(* CODESYS project opas-OCFB_IN-test-project

Project tree, tasks and I/O mapping:
  Device : CODESYS Control Win V3 x64, 3S - Smart Software Solutions GmbH, version 3.5.19.10
    application Application
      libraries: Standard, 3.5.18.0 (System); OPAS OCF Library, 1.0.0.0 (CODESYS Corporation)
      task MainTask (cyclic, interval t#20ms, priority 1) calls PLC_PRG
      program OCFBs [LD]
      program OCFBs_sim [LD]
      program PLC_PRG [ST]
      Sandbox/
        function block FB_FINAL_TEST [ST]
      SIM/
      visualisation Visualization
    SoftMotion General Axis Pool : SoftMotion General Axis Pool, 3S - Smart Software Solutions GmbH, version 4.11.0.0
    SoftMotion General Axis Pool : SoftMotion General Axis Pool, 3S - Smart Software Solutions GmbH, version 4.11.0.0
  text list GlobalTextList
*)

// Device/Application/PLC_PRG
PROGRAM PLC_PRG
VAR
	xAddConnection : BOOL;
	myAliasServerConnection : org_opengroup_opas_OCF.AliasServerConnection;
	fbFinal1 : FB_FINAL_TEST;
	fbFinal2 : FB_FINAL_TEST;
END_VAR

//OCFBs_sim();
OCFBs();

END_PROGRAM

// Device/Application/OCFBs_sim
PROGRAM OCFBs_sim
VAR
	xEnableAll : bool := true;
	tag1_OCFB_IN_SIM: org_opengroup_opas_OCF.OCFB_IN_SIM;
	tag2_OCFB_IN_SIM: org_opengroup_opas_OCF.OCFB_IN_SIM;
	tag3_OCFB_IN_SIM: org_opengroup_opas_OCF.OCFB_IN_SIM;
	tag4_OCFB_IN_SIM: org_opengroup_opas_OCF.OCFB_IN_SIM;
	tag5_OCFB_IN_SIM: org_opengroup_opas_OCF.OCFB_IN_SIM;
	tag6_OCFB_IN_SIM: org_opengroup_opas_OCF.OCFB_IN_SIM;
	tag7_OCFB_IN_SIM: org_opengroup_opas_OCF.OCFB_IN_SIM;
	
	xUtil1 : BOOL;
	xUtil2 : BOOL;
	xUtil3 : BOOL;
	xUtil4 : BOOL;
	iCount: UDINT;
END_VAR

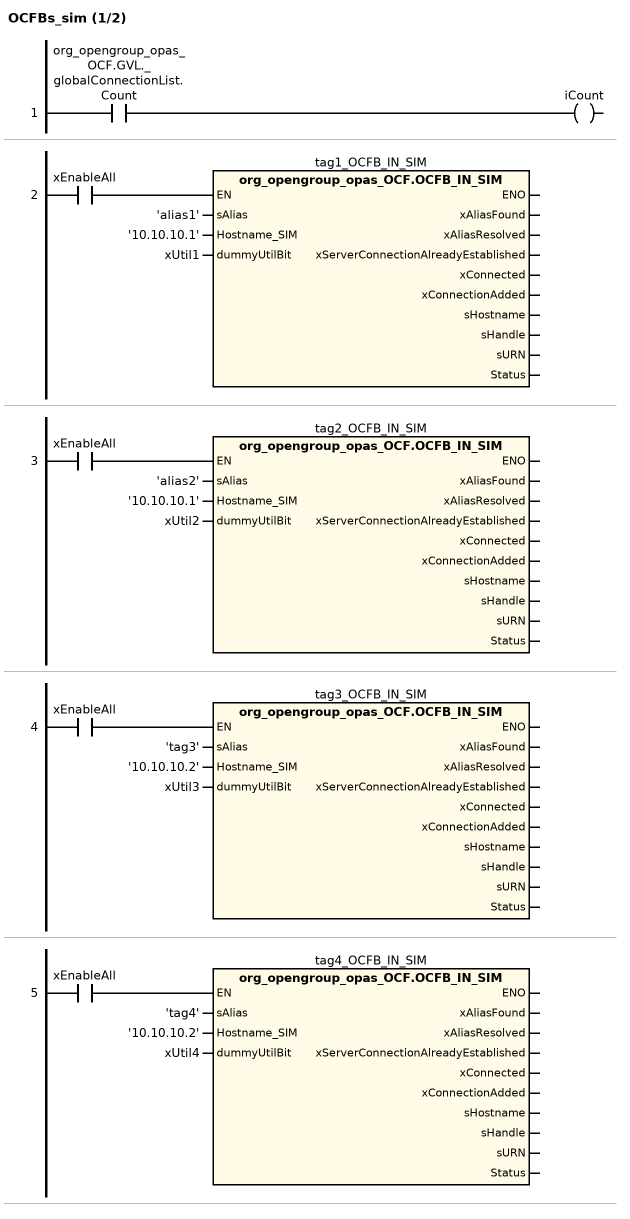
// NETWORK 1
iCount := org_opengroup_opas_OCF.GVL._globalConnectionList.Count;

// NETWORK 2
IF xEnableAll THEN
    tag1_OCFB_IN_SIM(sAlias := 'alias1', Hostname_SIM := '10.10.10.1', dummyUtilBit := xUtil1); // org_opengroup_opas_OCF.OCFB_IN_SIM
END_IF

// NETWORK 3
IF xEnableAll THEN
    tag2_OCFB_IN_SIM(sAlias := 'alias2', Hostname_SIM := '10.10.10.1', dummyUtilBit := xUtil2); // org_opengroup_opas_OCF.OCFB_IN_SIM
END_IF

// NETWORK 4
IF xEnableAll THEN
    tag3_OCFB_IN_SIM(sAlias := 'tag3', Hostname_SIM := '10.10.10.2', dummyUtilBit := xUtil3); // org_opengroup_opas_OCF.OCFB_IN_SIM
END_IF

// NETWORK 5
IF xEnableAll THEN
    tag4_OCFB_IN_SIM(sAlias := 'tag4', Hostname_SIM := '10.10.10.2', dummyUtilBit := xUtil4); // org_opengroup_opas_OCF.OCFB_IN_SIM
END_IF

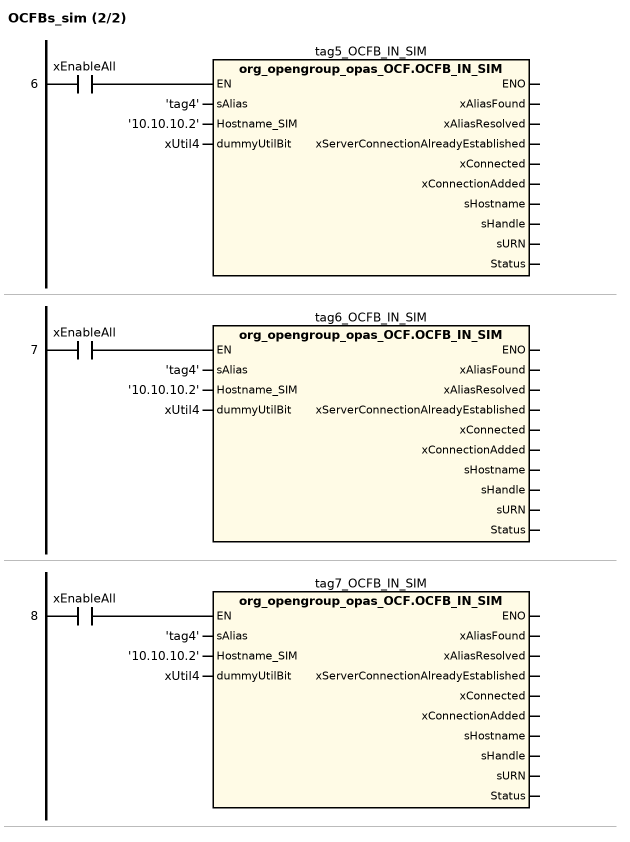
// NETWORK 6
IF xEnableAll THEN
    tag5_OCFB_IN_SIM(sAlias := 'tag4', Hostname_SIM := '10.10.10.2', dummyUtilBit := xUtil4); // org_opengroup_opas_OCF.OCFB_IN_SIM
END_IF

// NETWORK 7
IF xEnableAll THEN
    tag6_OCFB_IN_SIM(sAlias := 'tag4', Hostname_SIM := '10.10.10.2', dummyUtilBit := xUtil4); // org_opengroup_opas_OCF.OCFB_IN_SIM
END_IF

// NETWORK 8
IF xEnableAll THEN
    tag7_OCFB_IN_SIM(sAlias := 'tag4', Hostname_SIM := '10.10.10.2', dummyUtilBit := xUtil4); // org_opengroup_opas_OCF.OCFB_IN_SIM
END_IF

END_PROGRAM

// Device/Application/OCFBs
PROGRAM OCFBs
VAR
	xEnableAll : bool := true;
	tag1_OCFB_IN_SIM: org_opengroup_opas_OCF.OCFB_IN_LREAL;
	tag2_OCFB_IN_SIM: org_opengroup_opas_OCF.OCFB_IN_LREAL;
	//tag3_OCFB_IN_SIM: org_opengroup_opas_OCF.OCFB_IN_LREAL;
	//tag4_OCFB_IN_SIM: org_opengroup_opas_OCF.OCFB_IN_LREAL;
	//tag5_OCFB_IN_SIM: org_opengroup_opas_OCF.OCFB_IN_LREAL;
	//tag6_OCFB_IN_SIM: org_opengroup_opas_OCF.OCFB_IN_LREAL;
	//tag7_OCFB_IN_SIM: org_opengroup_opas_OCF.OCFB_IN_LREAL;
	
	xUtil1 : BOOL;
	xUtil2 : BOOL;
	xUtil3 : BOOL;
	xUtil4 : BOOL;
	iCount: UDINT;
	bEnable1: BOOL;
	bEnable2: BOOL;
END_VAR

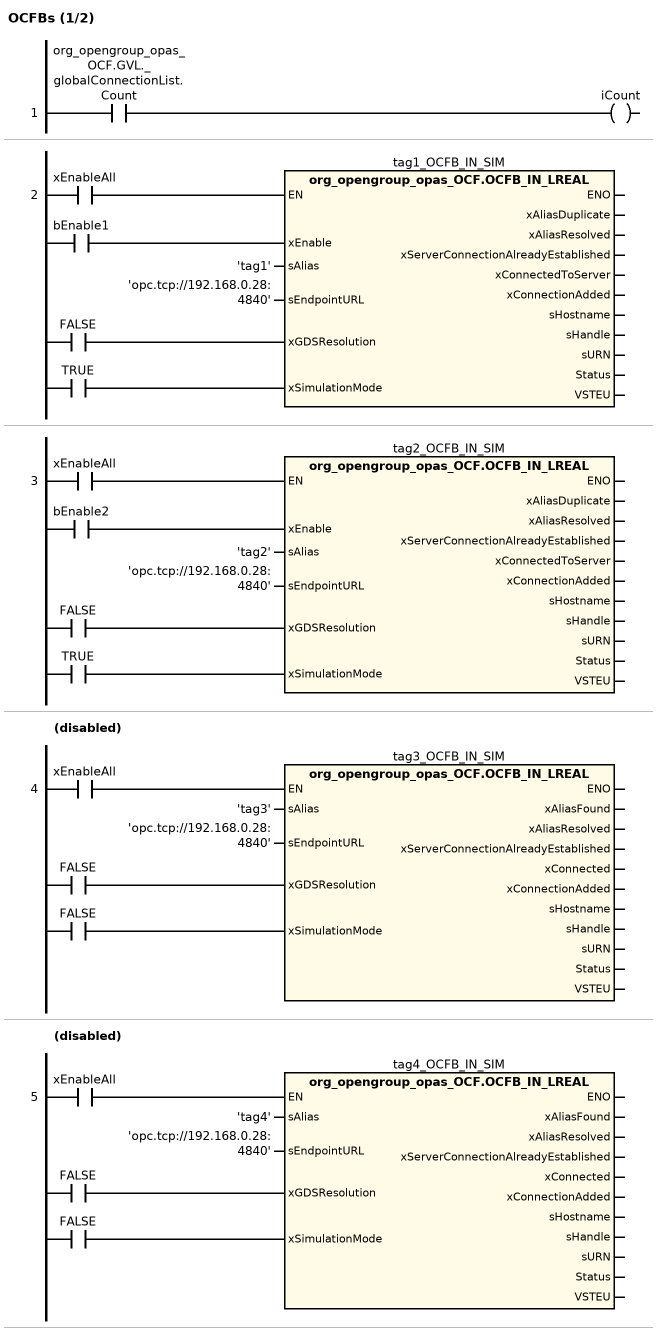
// NETWORK 1
iCount := org_opengroup_opas_OCF.GVL._globalConnectionList.Count;

// NETWORK 2
IF xEnableAll THEN
    tag1_OCFB_IN_SIM(
        xEnable := bEnable1,
        sAlias := 'tag1',
        sEndpointURL := 'opc.tcp://192.168.0.28:4840',
        xGDSResolution := FALSE,
        xSimulationMode := TRUE); // org_opengroup_opas_OCF.OCFB_IN_LREAL
END_IF

// NETWORK 3
IF xEnableAll THEN
    tag2_OCFB_IN_SIM(
        xEnable := bEnable2,
        sAlias := 'tag2',
        sEndpointURL := 'opc.tcp://192.168.0.28:4840',
        xGDSResolution := FALSE,
        xSimulationMode := TRUE); // org_opengroup_opas_OCF.OCFB_IN_LREAL
END_IF

// NETWORK 4 (disabled)
// IF xEnableAll THEN
//     tag3_OCFB_IN_SIM(
//         sAlias := 'tag3',
//         sEndpointURL := 'opc.tcp://192.168.0.28:4840',
//         xGDSResolution := FALSE,
//         xSimulationMode := FALSE); // org_opengroup_opas_OCF.OCFB_IN_LREAL
// END_IF

// NETWORK 5 (disabled)
// IF xEnableAll THEN
//     tag4_OCFB_IN_SIM(
//         sAlias := 'tag4',
//         sEndpointURL := 'opc.tcp://192.168.0.28:4840',
//         xGDSResolution := FALSE,
//         xSimulationMode := FALSE); // org_opengroup_opas_OCF.OCFB_IN_LREAL
// END_IF

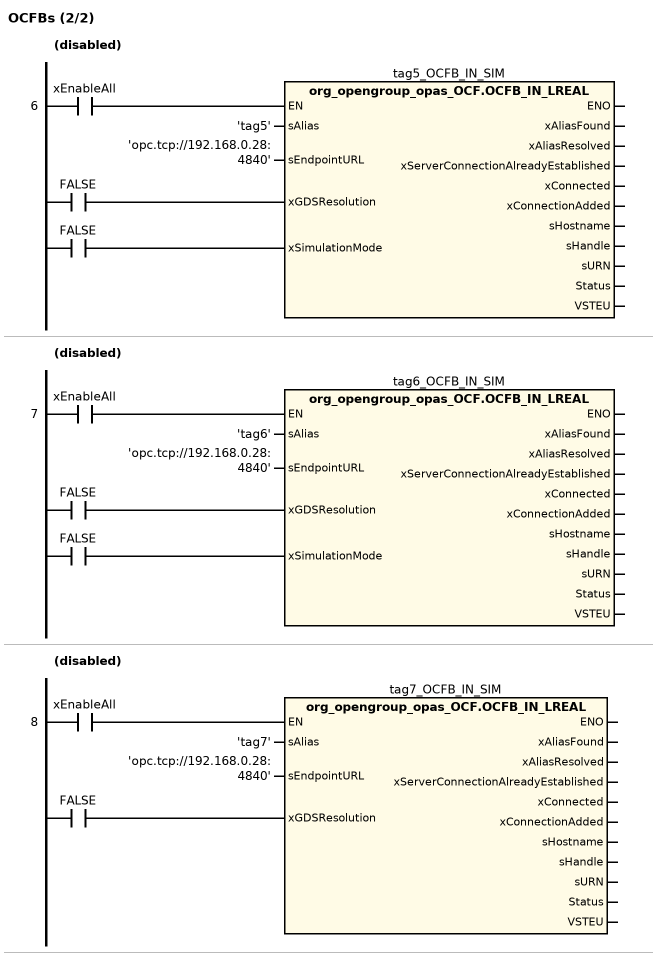
// NETWORK 6 (disabled)
// IF xEnableAll THEN
//     tag5_OCFB_IN_SIM(
//         sAlias := 'tag5',
//         sEndpointURL := 'opc.tcp://192.168.0.28:4840',
//         xGDSResolution := FALSE,
//         xSimulationMode := FALSE); // org_opengroup_opas_OCF.OCFB_IN_LREAL
// END_IF

// NETWORK 7 (disabled)
// IF xEnableAll THEN
//     tag6_OCFB_IN_SIM(
//         sAlias := 'tag6',
//         sEndpointURL := 'opc.tcp://192.168.0.28:4840',
//         xGDSResolution := FALSE,
//         xSimulationMode := FALSE); // org_opengroup_opas_OCF.OCFB_IN_LREAL
// END_IF

// NETWORK 8 (disabled)
// IF xEnableAll THEN
//     tag7_OCFB_IN_SIM(sAlias := 'tag7', sEndpointURL := 'opc.tcp://192.168.0.28:4840', xGDSResolution := FALSE); // org_opengroup_opas_OCF.OCFB_IN_LREAL
// END_IF

END_PROGRAM

// Device/Application/Sandbox/FB_FINAL_TEST
FUNCTION_BLOCK FINAL FB_FINAL_TEST
VAR_INPUT
	xEnable : BOOL;
END_VAR
VAR_OUTPUT
	xEnabled : bool;
END_VAR
VAR
END_VAR

xEnabled := xEnable;

END_FUNCTION_BLOCK

// Device/Application/Visualization
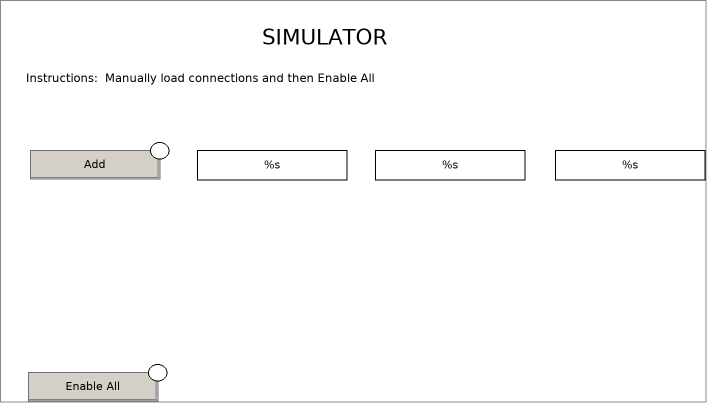
VISUALIZATION Visualization  // 707x403
    Group (28,364 139x37)
        Button (0,8 130x29), "Enable All"
            toggle OCFBs_sim.xEnableAll
        Ellipse (120,0 19x17), colour toggle: OCFBs_sim.xEnableAll
    Label (250,22 150x30), "SIMULATOR"
    Label (23,70 363x34), "Instructions: Manually load connections and then Enable All"
    Group (30,142 139x37)
        Button (0,8 130x29), "Add"
            tap PLC_PRG.xAddConnection
        Ellipse (120,0 19x17), colour toggle: PLC_PRG.xAddConnection
    Rectangle (197,150 150x30), "%s"
    Rectangle (375,150 150x30), "%s"
    Rectangle (555,150 150x30), "%s"
END_VISUALIZATION
